PROGRAM VelocityRide
VAR
	startVelocity: BOOL := FALSE;
	VelocityCounter: DINT;
	VelocityInterval: DINT := 2000;
	VelocityMmPerSecond: DINT := 5;
	
	state: INT := 0;
	
END_VAR

CASE state OF


0 :
	
	IF MAIN.dummy = 0 AND startVelocity  THEN
		state := 10;
	ELSIF MAIN.dummy = 1 AND startVelocity THEN
		state := 30;
	END_IF	
		
10 : 
			IF startVelocity THEN
				VelocityCounter := VelocityCounter + 1;
				IF VelocityCounter < VelocityInterval THEN
					link.xAxisVelocity := TO_DINT((VelocityMmPerSecond + 10 * 0) / 5 * 10000 * 60 );
					
				ELSIF VelocityCounter >= VelocityInterval AND VelocityCounter < VelocityInterval * 2 THEN
					link.xAxisVelocity := TO_DINT(-(VelocityMmPerSecond + 10 * 0) / 5 * 10000 * 60 );
					
				ELSIF VelocityCounter >= VelocityInterval*2 AND VelocityCounter < VelocityInterval*3 THEN
					link.xAxisVelocity := TO_DINT((VelocityMmPerSecond + 10 * 1) / 5 * 10000 * 60 );
 
				ELSIF VelocityCounter >= VelocityInterval*3 AND VelocityCounter < VelocityInterval*4 THEN
					link.xAxisVelocity := TO_DINT(-(VelocityMmPerSecond + 10 * 1) / 5 * 10000 * 60);
					
				ELSIF VelocityCounter >= VelocityInterval*4 AND VelocityCounter < VelocityInterval*5 THEN
					link.xAxisVelocity := TO_DINT((VelocityMmPerSecond + 10 * 2) / 5 * 10000 * 60 );
 
				ELSIF VelocityCounter >= VelocityInterval*5 AND VelocityCounter < VelocityInterval*6 THEN
					link.xAxisVelocity := TO_DINT(-(VelocityMmPerSecond + 10 * 2) / 5 * 10000 * 60);
					
				ELSIF VelocityCounter >= VelocityInterval*6 AND VelocityCounter < VelocityInterval*7 THEN
					link.xAxisVelocity := TO_DINT((VelocityMmPerSecond + 10 * 3) / 5 * 10000 * 60);
					
				ELSIF VelocityCounter >= VelocityInterval*7 AND VelocityCounter < VelocityInterval*8 THEN
					link.xAxisVelocity := TO_DINT(-(VelocityMmPerSecond + 10 * 3) / 5 * 10000 * 60);
					
				ELSIF VelocityCounter >= VelocityInterval*8 AND VelocityCounter < VelocityInterval*9 THEN
					link.xAxisVelocity := TO_DINT((VelocityMmPerSecond + 10 * 4) / 5 * 10000 * 60);
					
				ELSIF VelocityCounter >= VelocityInterval*9 AND VelocityCounter < VelocityInterval*10 THEN
					link.xAxisVelocity := TO_DINT(-(VelocityMmPerSecond + 10 * 4) / 5 * 10000 * 60);
					
				ELSIF VelocityCounter >= VelocityInterval*10 AND VelocityCounter < VelocityInterval*11 THEN
					link.xAxisVelocity := TO_DINT((VelocityMmPerSecond + 10 * 5) / 5 * 10000 * 60);
					
				ELSIF VelocityCounter >= VelocityInterval*11 AND VelocityCounter < VelocityInterval*12 THEN
					link.xAxisVelocity := TO_DINT(-(VelocityMmPerSecond + 10 * 5) / 5 * 10000 * 60);
					
				ELSIF VelocityCounter >= VelocityInterval*12 AND VelocityCounter < VelocityInterval*13 THEN
					link.xAxisVelocity := TO_DINT((VelocityMmPerSecond + 10 * 6) / 5 * 10000 * 60);
					
				ELSIF VelocityCounter >= VelocityInterval*13 AND VelocityCounter < VelocityInterval*14 THEN
					link.xAxisVelocity := TO_DINT(-(VelocityMmPerSecond + 10 * 6) / 5 * 10000 * 60);
					
				ELSIF VelocityCounter >= VelocityInterval*14 AND VelocityCounter < VelocityInterval*15 THEN
					link.xAxisVelocity := TO_DINT((VelocityMmPerSecond + 10 * 7) / 5 * 10000 * 60);
					
				ELSIF VelocityCounter >= VelocityInterval*15 AND VelocityCounter < VelocityInterval*16 THEN
					link.xAxisVelocity := TO_DINT(-(VelocityMmPerSecond + 10 * 7) / 5 * 10000 * 60);
					
				ELSIF VelocityCounter >= VelocityInterval*16 AND VelocityCounter < VelocityInterval*17 THEN
					link.xAxisVelocity := TO_DINT((VelocityMmPerSecond + 10 * 8) / 5 * 10000 * 60);
					
				ELSIF VelocityCounter >= VelocityInterval*17 AND VelocityCounter < VelocityInterval*18 THEN
					link.xAxisVelocity := TO_DINT(-(VelocityMmPerSecond + 10 * 8) / 5 * 10000 * 60);
					
				ELSIF VelocityCounter >= VelocityInterval*18 AND VelocityCounter < VelocityInterval*19 THEN
					link.xAxisVelocity := TO_DINT((VelocityMmPerSecond + 10 * 9) / 5 * 10000 * 60);
					
				ELSIF VelocityCounter >= VelocityInterval*19 AND VelocityCounter < VelocityInterval*20 THEN
					link.xAxisVelocity := TO_DINT(-(VelocityMmPerSecond + 10 * 9) / 5 * 10000 * 60);
					
				ELSIF VelocityCounter >= VelocityInterval*20 AND VelocityCounter < VelocityInterval*21 THEN
					link.xAxisVelocity := TO_DINT((VelocityMmPerSecond + 10 * 10) / 5 * 10000 * 60);
					
				ELSIF VelocityCounter >= VelocityInterval*21 AND VelocityCounter < VelocityInterval*22 THEN
					link.xAxisVelocity := TO_DINT(-(VelocityMmPerSecond + 10 * 10) / 5 * 10000 * 60);
					
				ELSIF VelocityCounter >= VelocityInterval*22 THEN
					link.xAxisVelocity := 0;
					startVelocity := 0;
					state := 60;
					
				END_IF
			ELSE
				state := 60;
			END_IF
			
30 : 
			IF startVelocity THEN
				VelocityCounter := VelocityCounter + 1;
				IF VelocityCounter < VelocityInterval THEN
					link.yAxisVelocity := TO_DINT((VelocityMmPerSecond + 10 * 0) / 5 * 10000 * 60 );
					
				ELSIF VelocityCounter >= VelocityInterval AND VelocityCounter < VelocityInterval * 2 THEN
					link.yAxisVelocity := TO_DINT(-(VelocityMmPerSecond + 10 * 0) / 5 * 10000 * 60 );
					
				ELSIF VelocityCounter >= VelocityInterval*2 AND VelocityCounter < VelocityInterval*3 THEN
					link.yAxisVelocity := TO_DINT((VelocityMmPerSecond + 10 * 1) / 5 * 10000 * 60 );
 
				ELSIF VelocityCounter >= VelocityInterval*3 AND VelocityCounter < VelocityInterval*4 THEN
					link.yAxisVelocity := TO_DINT(-(VelocityMmPerSecond + 10 * 1) / 5 * 10000 * 60);
					
				ELSIF VelocityCounter >= VelocityInterval*4 AND VelocityCounter < VelocityInterval*5 THEN
					link.yAxisVelocity := TO_DINT((VelocityMmPerSecond + 10 * 2) / 5 * 10000 * 60 );
 
				ELSIF VelocityCounter >= VelocityInterval*5 AND VelocityCounter < VelocityInterval*6 THEN
					link.yAxisVelocity := TO_DINT(-(VelocityMmPerSecond + 10 * 2) / 5 * 10000 * 60);
					
				ELSIF VelocityCounter >= VelocityInterval*6 AND VelocityCounter < VelocityInterval*7 THEN
					link.yAxisVelocity := TO_DINT((VelocityMmPerSecond + 10 * 3) / 5 * 10000 * 60);
					
				ELSIF VelocityCounter >= VelocityInterval*7 AND VelocityCounter < VelocityInterval*8 THEN
					link.yAxisVelocity := TO_DINT(-(VelocityMmPerSecond + 10 * 3) / 5 * 10000 * 60);
					
				ELSIF VelocityCounter >= VelocityInterval*8 AND VelocityCounter < VelocityInterval*9 THEN
					link.yAxisVelocity := TO_DINT((VelocityMmPerSecond + 10 * 4) / 5 * 10000 * 60);
					
				ELSIF VelocityCounter >= VelocityInterval*9 AND VelocityCounter < VelocityInterval*10 THEN
					link.yAxisVelocity := TO_DINT(-(VelocityMmPerSecond + 10 * 4) / 5 * 10000 * 60);
					
				ELSIF VelocityCounter >= VelocityInterval*10 AND VelocityCounter < VelocityInterval*11 THEN
					link.yAxisVelocity := TO_DINT((VelocityMmPerSecond + 10 * 5) / 5 * 10000 * 60);
					
				ELSIF VelocityCounter >= VelocityInterval*11 AND VelocityCounter < VelocityInterval*12 THEN
					link.yAxisVelocity := TO_DINT(-(VelocityMmPerSecond + 10 * 5) / 5 * 10000 * 60);
					
				ELSIF VelocityCounter >= VelocityInterval*12 AND VelocityCounter < VelocityInterval*13 THEN
					link.yAxisVelocity := TO_DINT((VelocityMmPerSecond + 10 * 6) / 5 * 10000 * 60);
					
				ELSIF VelocityCounter >= VelocityInterval*13 AND VelocityCounter < VelocityInterval*14 THEN
					link.yAxisVelocity := TO_DINT(-(VelocityMmPerSecond + 10 * 6) / 5 * 10000 * 60);
					
				ELSIF VelocityCounter >= VelocityInterval*14 AND VelocityCounter < VelocityInterval*15 THEN
					link.yAxisVelocity := TO_DINT((VelocityMmPerSecond + 10 * 7) / 5 * 10000 * 60);
					
				ELSIF VelocityCounter >= VelocityInterval*15 AND VelocityCounter < VelocityInterval*16 THEN
					link.yAxisVelocity := TO_DINT(-(VelocityMmPerSecond + 10 * 7) / 5 * 10000 * 60);
					
				ELSIF VelocityCounter >= VelocityInterval*16 AND VelocityCounter < VelocityInterval*17 THEN
					link.yAxisVelocity := TO_DINT((VelocityMmPerSecond + 10 * 8) / 5 * 10000 * 60);
					
				ELSIF VelocityCounter >= VelocityInterval*17 AND VelocityCounter < VelocityInterval*18 THEN
					link.yAxisVelocity := TO_DINT(-(VelocityMmPerSecond + 10 * 8) / 5 * 10000 * 60);
					
				ELSIF VelocityCounter >= VelocityInterval*18 AND VelocityCounter < VelocityInterval*19 THEN
					link.yAxisVelocity := TO_DINT((VelocityMmPerSecond + 10 * 9) / 5 * 10000 * 60);
					
				ELSIF VelocityCounter >= VelocityInterval*19 AND VelocityCounter < VelocityInterval*20 THEN
					link.yAxisVelocity := TO_DINT(-(VelocityMmPerSecond + 10 * 9) / 5 * 10000 * 60);
					
				ELSIF VelocityCounter >= VelocityInterval*20 AND VelocityCounter < VelocityInterval*21 THEN
					link.yAxisVelocity := TO_DINT((VelocityMmPerSecond + 10 * 10) / 5 * 10000 * 60);
					
				ELSIF VelocityCounter >= VelocityInterval*21 AND VelocityCounter < VelocityInterval*22 THEN
					link.yAxisVelocity := TO_DINT(-(VelocityMmPerSecond + 10 * 10) / 5 * 10000 * 60);
					
				ELSIF VelocityCounter >= VelocityInterval*22 THEN
					link.yAxisVelocity := 0;
					startVelocity := 0;
					state := 60;
					
				END_IF
			ELSE
				state := 60;
			END_IF
			
60 :
	startVelocity:= FALSE;
	state :=0;
	VelocityCounter := 0;
END_CASE

END_PROGRAM

(* stored: Version 1.1.0.1, ProductVersion 3.1.4024.9
   POU VelocityRide: Id {333edcd8-7d23-44a5-9a35-7ff3ff5d622a}, SpecialFunc None *)
